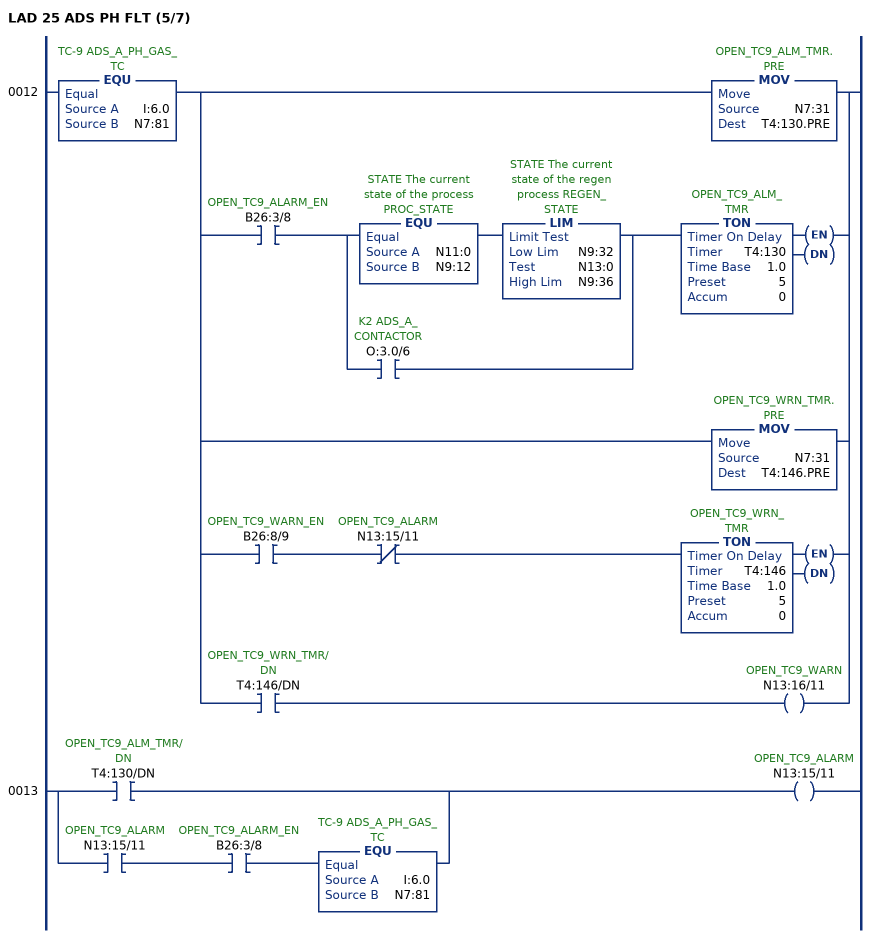
% Rung: 12 %
SOR EQU I:6.0 N7:81 BST MOV N7:31 T4:130.PRE NXB XIC B26:3/8 BST EQU N11:0 N9:12 LIM N9:32 N13:0 N9:36 NXB XIC O:3.0/6 BND TON T4:130 1.0 5 0 NXB MOV N7:31 T4:146.PRE NXB XIC B26:8/9 XIO N13:15/11 TON T4:146 1.0 5 0 NXB XIC T4:146/DN OTE N13:16/11 BND EOR
%   I:6.0  ADS_A_PH_GAS_TC  "TC-9" %
%   N7:81  TC_OPEN_SP  "CONFIG The value read by an open TC input" %
%   N7:31  OPEN_TC_DLY %
%   T4:130  OPEN_TC9_ALM_TMR %
%   B26:3/8  OPEN_TC9_ALARM_EN %
%   N11:0  PROC_STATE  "STATE The current state of the process" %
%   N9:12  PROC_PFY_B_REG_A  "STATE Process Purify B" %
%   N9:32  REGEN_VENT  "STATE Regen Vent" %
%   N13:0  REGEN_STATE  "STATE The current state of the regen process" %
%   N9:36  REGEN_COOL  "STATE Regen Cool" %
%   O:3.0/6  ADS_A_CONTACTOR  "K2" %
%   T4:146  OPEN_TC9_WRN_TMR %
%   B26:8/9  OPEN_TC9_WARN_EN %
%   N13:15/11  OPEN_TC9_ALARM %
%   N13:16/11  OPEN_TC9_WARN %
% Rung: 13 %
SOR BST XIC T4:130/DN NXB XIC N13:15/11 XIC B26:3/8 EQU I:6.0 N7:81 BND OTE N13:15/11 EOR
%   T4:130  OPEN_TC9_ALM_TMR %
%   N13:15/11  OPEN_TC9_ALARM %
%   B26:3/8  OPEN_TC9_ALARM_EN %
%   I:6.0  ADS_A_PH_GAS_TC  "TC-9" %
%   N7:81  TC_OPEN_SP  "CONFIG The value read by an open TC input" %

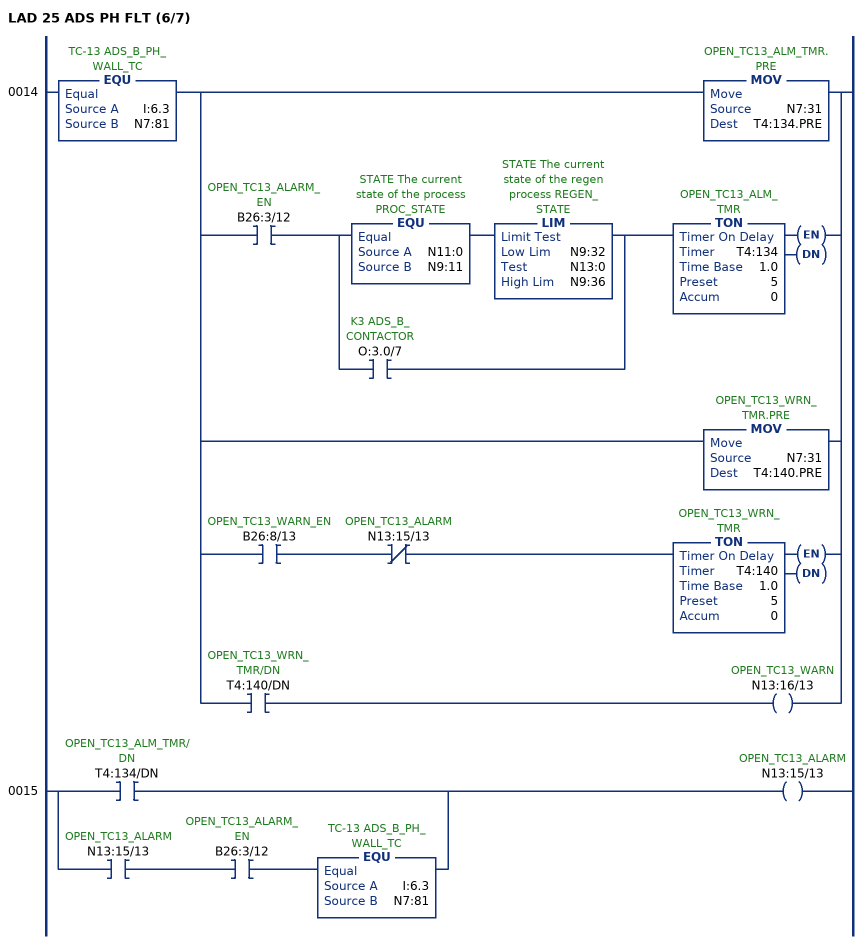
% Rung: 14 %
SOR EQU I:6.3 N7:81 BST MOV N7:31 T4:134.PRE NXB XIC B26:3/12 BST EQU N11:0 N9:11 LIM N9:32 N13:0 N9:36 NXB XIC O:3.0/7 BND TON T4:134 1.0 5 0 NXB MOV N7:31 T4:140.PRE NXB XIC B26:8/13 XIO N13:15/13 TON T4:140 1.0 5 0 NXB XIC T4:140/DN OTE N13:16/13 BND EOR
%   I:6.3  ADS_B_PH_WALL_TC  "TC-13" %
%   N7:81  TC_OPEN_SP  "CONFIG The value read by an open TC input" %
%   N7:31  OPEN_TC_DLY %
%   T4:134  OPEN_TC13_ALM_TMR %
%   B26:3/12  OPEN_TC13_ALARM_EN %
%   N11:0  PROC_STATE  "STATE The current state of the process" %
%   N9:11  PROC_PFY_A_REG_B  "STATE Process Purify A" %
%   N9:32  REGEN_VENT  "STATE Regen Vent" %
%   N13:0  REGEN_STATE  "STATE The current state of the regen process" %
%   N9:36  REGEN_COOL  "STATE Regen Cool" %
%   O:3.0/7  ADS_B_CONTACTOR  "K3" %
%   T4:140  OPEN_TC13_WRN_TMR %
%   B26:8/13  OPEN_TC13_WARN_EN %
%   N13:15/13  OPEN_TC13_ALARM %
%   N13:16/13  OPEN_TC13_WARN %
% Rung: 15 %
SOR BST XIC T4:134/DN NXB XIC N13:15/13 XIC B26:3/12 EQU I:6.3 N7:81 BND OTE N13:15/13 EOR
%   T4:134  OPEN_TC13_ALM_TMR %
%   N13:15/13  OPEN_TC13_ALARM %
%   B26:3/12  OPEN_TC13_ALARM_EN %
%   I:6.3  ADS_B_PH_WALL_TC  "TC-13" %
%   N7:81  TC_OPEN_SP  "CONFIG The value read by an open TC input" %

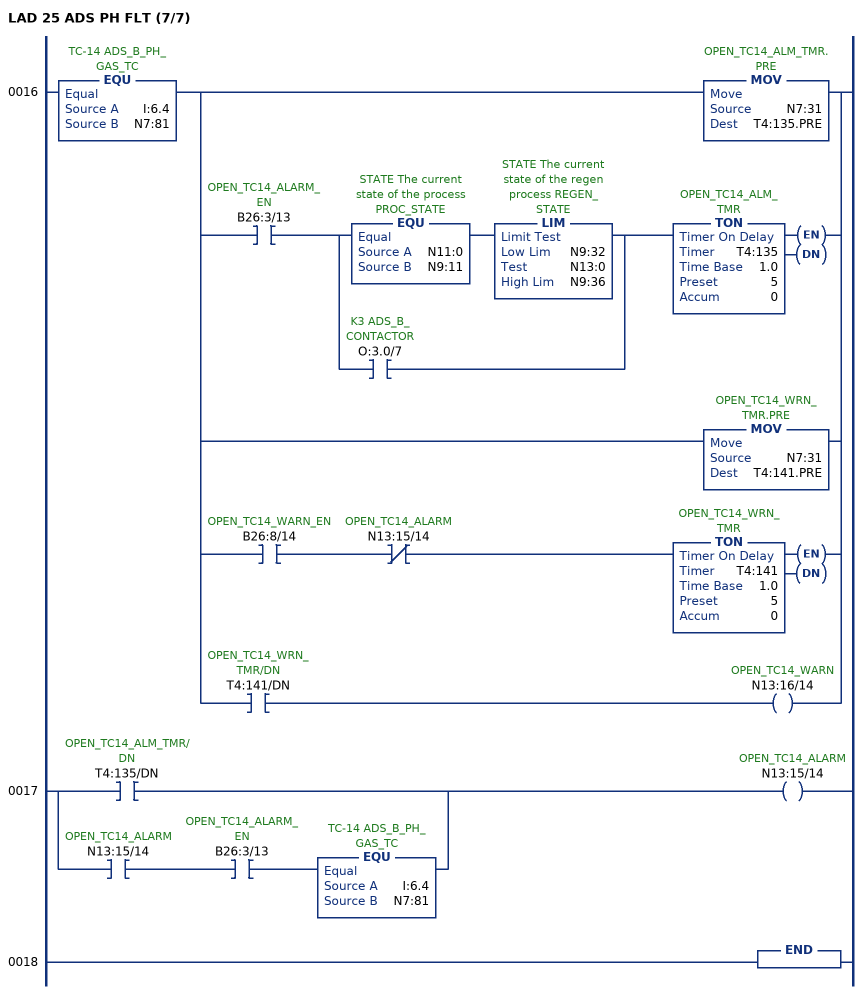
% Rung: 16 %
SOR EQU I:6.4 N7:81 BST MOV N7:31 T4:135.PRE NXB XIC B26:3/13 BST EQU N11:0 N9:11 LIM N9:32 N13:0 N9:36 NXB XIC O:3.0/7 BND TON T4:135 1.0 5 0 NXB MOV N7:31 T4:141.PRE NXB XIC B26:8/14 XIO N13:15/14 TON T4:141 1.0 5 0 NXB XIC T4:141/DN OTE N13:16/14 BND EOR
%   I:6.4  ADS_B_PH_GAS_TC  "TC-14" %
%   N7:81  TC_OPEN_SP  "CONFIG The value read by an open TC input" %
%   N7:31  OPEN_TC_DLY %
%   T4:135  OPEN_TC14_ALM_TMR %
%   B26:3/13  OPEN_TC14_ALARM_EN %
%   N11:0  PROC_STATE  "STATE The current state of the process" %
%   N9:11  PROC_PFY_A_REG_B  "STATE Process Purify A" %
%   N9:32  REGEN_VENT  "STATE Regen Vent" %
%   N13:0  REGEN_STATE  "STATE The current state of the regen process" %
%   N9:36  REGEN_COOL  "STATE Regen Cool" %
%   O:3.0/7  ADS_B_CONTACTOR  "K3" %
%   T4:141  OPEN_TC14_WRN_TMR %
%   B26:8/14  OPEN_TC14_WARN_EN %
%   N13:15/14  OPEN_TC14_ALARM %
%   N13:16/14  OPEN_TC14_WARN %
% Rung: 17 %
SOR BST XIC T4:135/DN NXB XIC N13:15/14 XIC B26:3/13 EQU I:6.4 N7:81 BND OTE N13:15/14 EOR
%   T4:135  OPEN_TC14_ALM_TMR %
%   N13:15/14  OPEN_TC14_ALARM %
%   B26:3/13  OPEN_TC14_ALARM_EN %
%   I:6.4  ADS_B_PH_GAS_TC  "TC-14" %
%   N7:81  TC_OPEN_SP  "CONFIG The value read by an open TC input" %
% Rung: 18 %
SOR END EOR

LADDER 26 "GETTER"
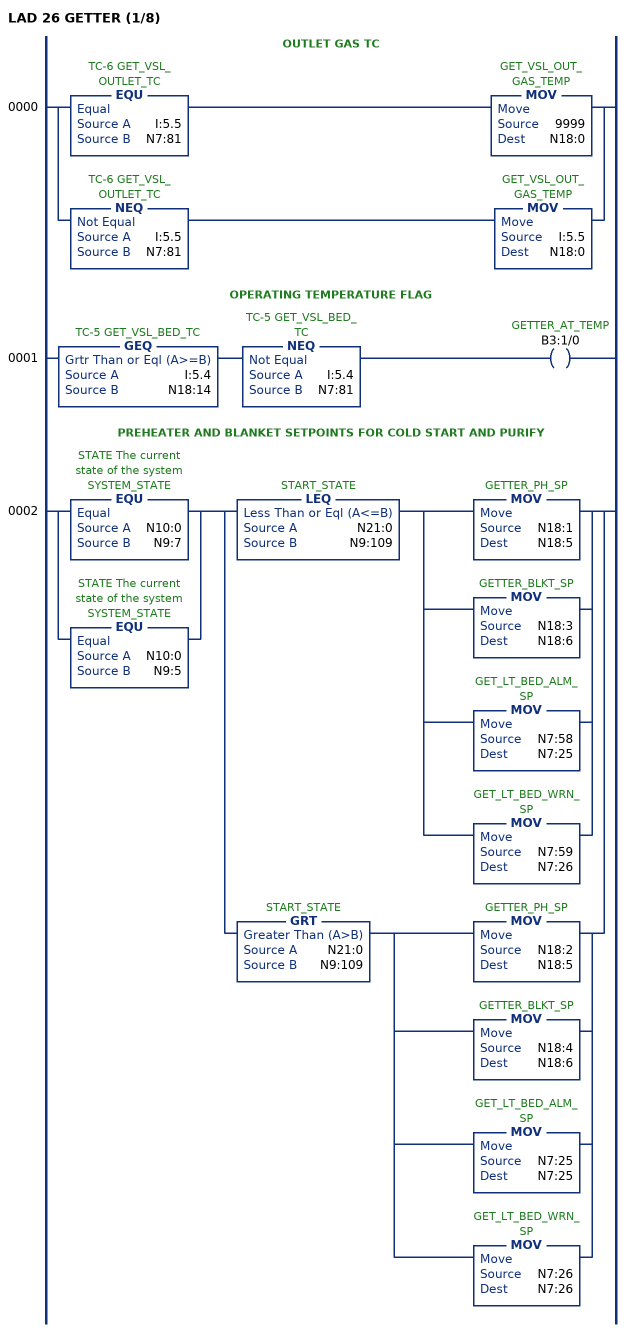
% Rung: 0 %
% TITLE: OUTLET GAS TC %
SOR BST EQU I:5.5 N7:81 MOV 9999 N18:0 NXB NEQ I:5.5 N7:81 MOV I:5.5 N18:0 BND EOR
%   I:5.5  GET_VSL_OUTLET_TC  "TC-6" %
%   N7:81  TC_OPEN_SP  "CONFIG The value read by an open TC input" %
%   N18:0  GET_VSL_OUT_GAS_TEMP %
% Rung: 1 %
% TITLE: OPERATING TEMPERATURE FLAG %
SOR GEQ I:5.4 N18:14 NEQ I:5.4 N7:81 OTE B3:1/0 EOR
%   I:5.4  GET_VSL_BED_TC  "TC-5" %
%   N18:14  GETTER_OPERATING_TMP %
%   N7:81  TC_OPEN_SP  "CONFIG The value read by an open TC input" %
%   B3:1/0  GETTER_AT_TEMP %
% Rung: 2 %
% TITLE: PREHEATER AND BLANKET SETPOINTS FOR COLD START AND PURIFY %
SOR BST EQU N10:0 N9:7 NXB EQU N10:0 N9:5 BND BST LEQ N21:0 N9:109 BST MOV N18:1 N18:5 NXB MOV N18:3 N18:6 NXB MOV N7:58 N7:25 NXB MOV N7:59 N7:26 BND NXB GRT N21:0 N9:109 BST MOV N18:2 N18:5 NXB MOV N18:4 N18:6 NXB MOV N7:25 N7:25 NXB MOV N7:26 N7:26 BND BND EOR
%   N10:0  SYSTEM_STATE  "STATE The current state of the system" %
%   N9:7  SYSTEM_COLD_START %
%   N9:5  SYSTEM_QUICK_START %
%   N21:0  START_STATE %
%   N9:109  START_BKFL_2 %
%   N18:1  GETTER_COLD_PH_SP %
%   N18:5  GETTER_PH_SP %
%   N18:3  GETTER_COLD_BLKT_SP %
%   N18:6  GETTER_BLKT_SP %
%   N7:58  GET_LT_BED_ST_ALM_SP %
%   N7:25  GET_LT_BED_ALM_SP %
%   N7:59  GET_LT_BED_ST_WRN_SP %
%   N7:26  GET_LT_BED_WRN_SP %
%   N18:2  GETTER_PFY_PH_SP %
%   N18:4  GETTER_PFY_BLKT_SP %

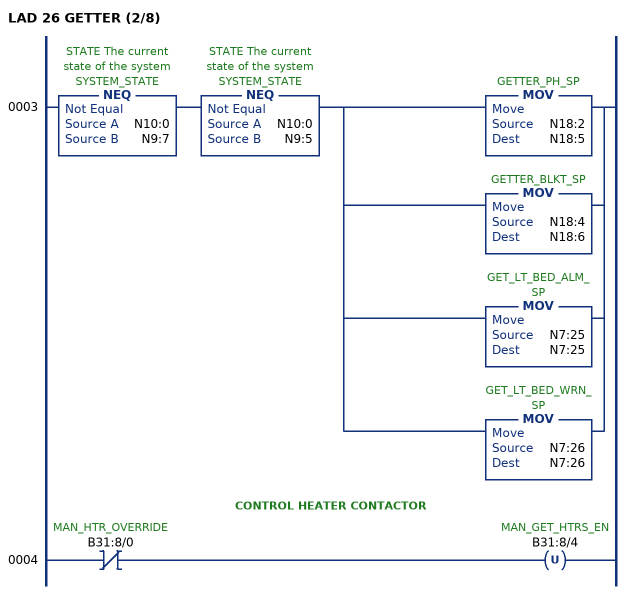
% Rung: 3 %
SOR NEQ N10:0 N9:7 NEQ N10:0 N9:5 BST MOV N18:2 N18:5 NXB MOV N18:4 N18:6 NXB MOV N7:25 N7:25 NXB MOV N7:26 N7:26 BND EOR
%   N10:0  SYSTEM_STATE  "STATE The current state of the system" %
%   N9:7  SYSTEM_COLD_START %
%   N9:5  SYSTEM_QUICK_START %
%   N18:2  GETTER_PFY_PH_SP %
%   N18:5  GETTER_PH_SP %
%   N18:4  GETTER_PFY_BLKT_SP %
%   N18:6  GETTER_BLKT_SP %
%   N7:25  GET_LT_BED_ALM_SP %
%   N7:26  GET_LT_BED_WRN_SP %
% Rung: 4 %
% TITLE: CONTROL HEATER CONTACTOR %
SOR XIO B31:8/0 OTU B31:8/4 EOR
%   B31:8/0  MAN_HTR_OVERRIDE %
%   B31:8/4  MAN_GET_HTRS_EN %

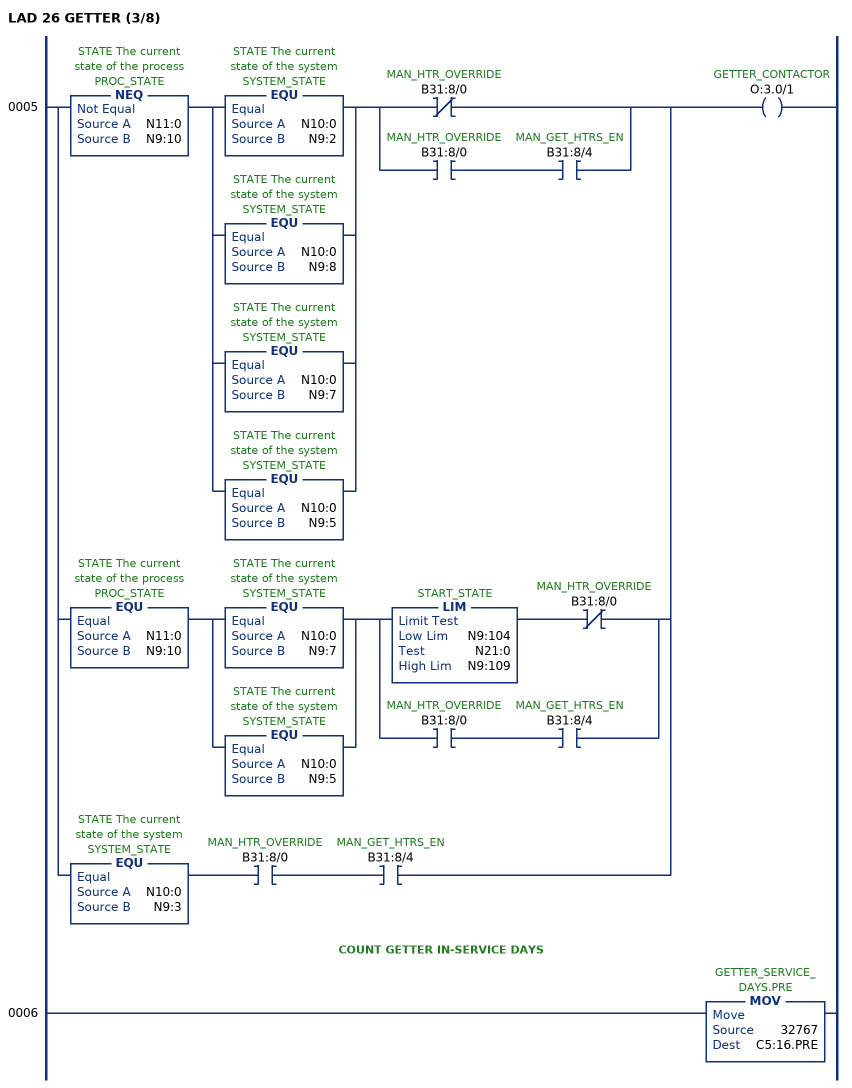
% Rung: 5 %
SOR BST NEQ N11:0 N9:10 BST EQU N10:0 N9:2 NXB EQU N10:0 N9:8 NXB EQU N10:0 N9:7 NXB EQU N10:0 N9:5 BND BST XIO B31:8/0 NXB XIC B31:8/0 XIC B31:8/4 BND NXB EQU N11:0 N9:10 BST EQU N10:0 N9:7 NXB EQU N10:0 N9:5 BND BST LIM N9:104 N21:0 N9:109 XIO B31:8/0 NXB XIC B31:8/0 XIC B31:8/4 BND NXB EQU N10:0 N9:3 XIC B31:8/0 XIC B31:8/4 BND OTE O:3.0/1 EOR
%   N11:0  PROC_STATE  "STATE The current state of the process" %
%   N9:10  PROC_STANDBY  "STATE Process Standby" %
%   N10:0  SYSTEM_STATE  "STATE The current state of the system" %
%   N9:2  SYSTEM_PROCESS  "STATE System Process" %
%   N9:8  SYSTEM_SUPPLEMENTAL %
%   N9:7  SYSTEM_COLD_START %
%   N9:5  SYSTEM_QUICK_START %
%   B31:8/0  MAN_HTR_OVERRIDE %
%   B31:8/4  MAN_GET_HTRS_EN %
%   N9:104  START_HEAT_GETTER %
%   N21:0  START_STATE %
%   N9:109  START_BKFL_2 %
%   N9:3  SYSTEM_MANUAL  "STATE System Manual" %
%   O:3.0/1  GETTER_CONTACTOR %
% Rung: 6 %
% TITLE: COUNT GETTER IN-SERVICE DAYS %
SOR MOV 32767 C5:16.PRE EOR
%   C5:16  GETTER_SERVICE_DAYS %

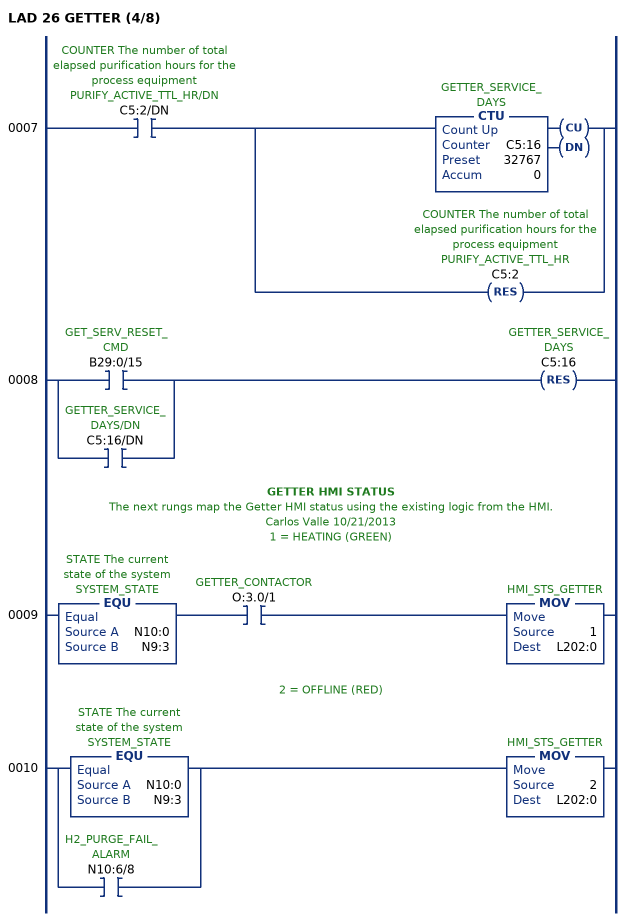
% Rung: 7 %
SOR XIC C5:2/DN BST CTU C5:16 32767 0 NXB RES C5:2 BND EOR
%   C5:2  PURIFY_ACTIVE_TTL_HR  "COUNTER The number of total elapsed purification hours for the process equipment" %
%   C5:16  GETTER_SERVICE_DAYS %
% Rung: 8 %
SOR BST XIC B29:0/15 NXB XIC C5:16/DN BND RES C5:16 EOR
%   B29:0/15  GET_SERV_RESET_CMD %
%   C5:16  GETTER_SERVICE_DAYS %
% Rung: 9 %
% TITLE: GETTER HMI STATUS %
% The next rungs map the Getter HMI status using the existing logic from the HMI.
% Carlos Valle 10/21/2013
% 1 = HEATING (GREEN) %
SOR EQU N10:0 N9:3 XIC O:3.0/1 MOV 1 L202:0 EOR
%   N10:0  SYSTEM_STATE  "STATE The current state of the system" %
%   N9:3  SYSTEM_MANUAL  "STATE System Manual" %
%   O:3.0/1  GETTER_CONTACTOR %
%   L202:0  HMI_STS_GETTER %
% Rung: 10 %
% 2 = OFFLINE (RED) %
SOR BST EQU N10:0 N9:3 NXB XIC N10:6/8 BND MOV 2 L202:0 EOR
%   N10:0  SYSTEM_STATE  "STATE The current state of the system" %
%   N9:3  SYSTEM_MANUAL  "STATE System Manual" %
%   N10:6/8  H2_PURGE_FAIL_ALARM %
%   L202:0  HMI_STS_GETTER %

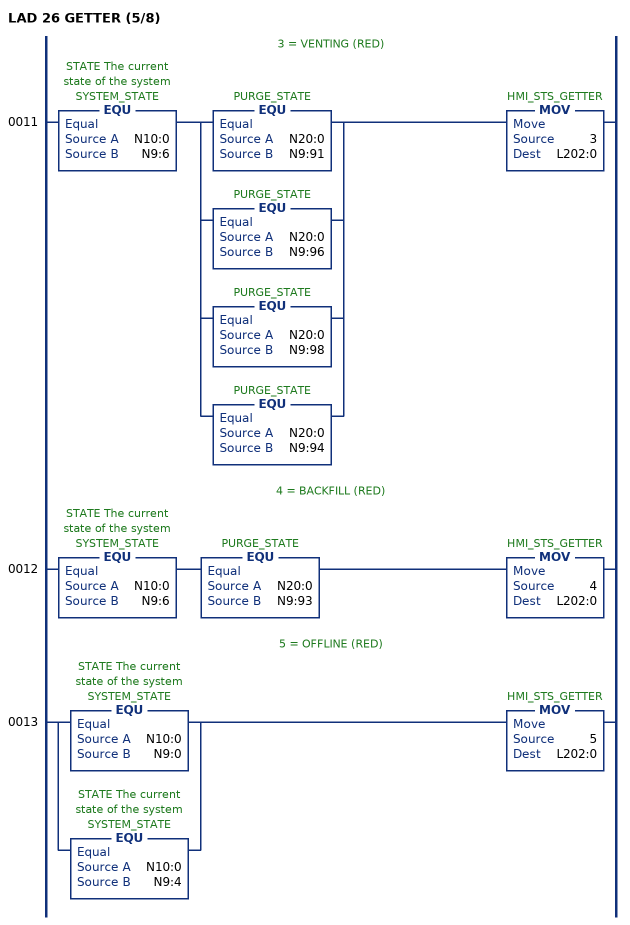
% Rung: 11 %
% 3 = VENTING (RED) %
SOR EQU N10:0 N9:6 BST EQU N20:0 N9:91 NXB EQU N20:0 N9:96 NXB EQU N20:0 N9:98 NXB EQU N20:0 N9:94 BND MOV 3 L202:0 EOR
%   N10:0  SYSTEM_STATE  "STATE The current state of the system" %
%   N9:6  SYSTEM_PURGE %
%   N20:0  PURGE_STATE %
%   N9:91  PURGE_INIT_VENT %
%   N9:96  PURGE_VENT_GETTER %
%   N9:98  PURGE_VENT_GET_2 %
%   N9:94  PURGE_FINAL_VENT %
%   L202:0  HMI_STS_GETTER %
% Rung: 12 %
% 4 = BACKFILL (RED) %
SOR EQU N10:0 N9:6 EQU N20:0 N9:93 MOV 4 L202:0 EOR
%   N10:0  SYSTEM_STATE  "STATE The current state of the system" %
%   N9:6  SYSTEM_PURGE %
%   N20:0  PURGE_STATE %
%   N9:93  PURGE_BACKFILL %
%   L202:0  HMI_STS_GETTER %
% Rung: 13 %
% 5 = OFFLINE (RED) %
SOR BST EQU N10:0 N9:0 NXB EQU N10:0 N9:4 BND MOV 5 L202:0 EOR
%   N10:0  SYSTEM_STATE  "STATE The current state of the system" %
%   N9:0  SYSTEM_OFFLINE %
%   N9:4  SYSTEM_ALARM  "STATE System Alarm" %
%   L202:0  HMI_STS_GETTER %

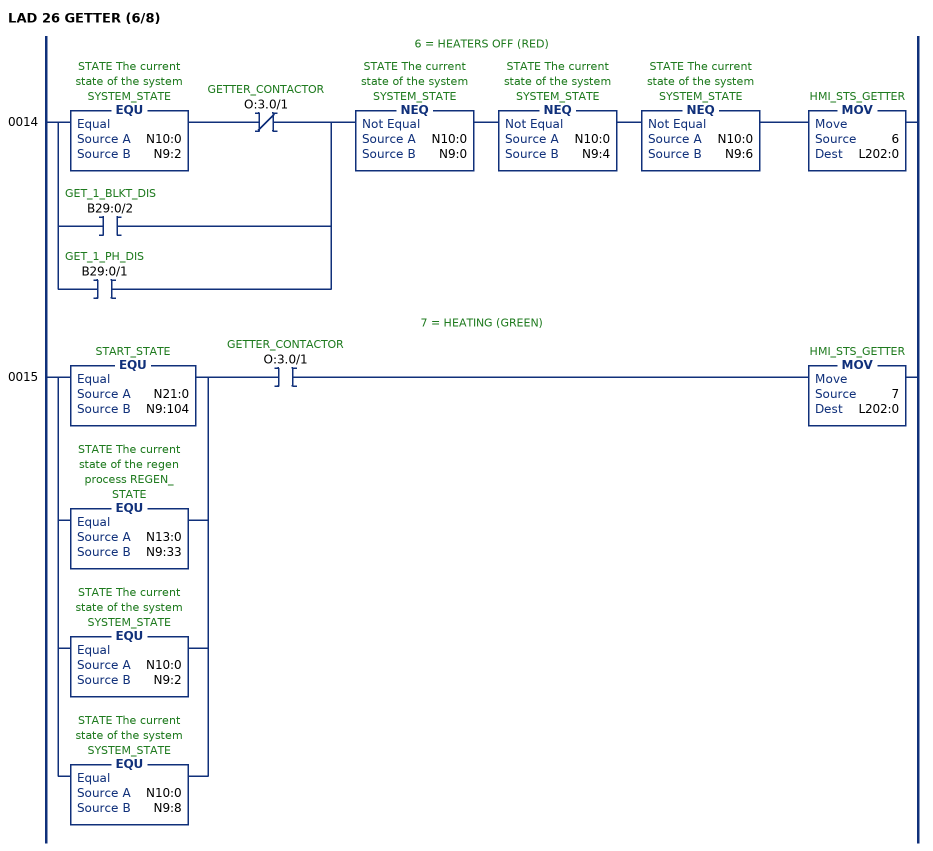
% Rung: 14 %
% 6 = HEATERS OFF (RED) %
SOR BST EQU N10:0 N9:2 XIO O:3.0/1 NXB XIC B29:0/2 NXB XIC B29:0/1 BND NEQ N10:0 N9:0 NEQ N10:0 N9:4 NEQ N10:0 N9:6 MOV 6 L202:0 EOR
%   N10:0  SYSTEM_STATE  "STATE The current state of the system" %
%   N9:2  SYSTEM_PROCESS  "STATE System Process" %
%   O:3.0/1  GETTER_CONTACTOR %
%   B29:0/2  GET_1_BLKT_DIS %
%   B29:0/1  GET_1_PH_DIS %
%   N9:0  SYSTEM_OFFLINE %
%   N9:4  SYSTEM_ALARM  "STATE System Alarm" %
%   N9:6  SYSTEM_PURGE %
%   L202:0  HMI_STS_GETTER %
% Rung: 15 %
% 7 = HEATING (GREEN) %
SOR BST EQU N21:0 N9:104 NXB EQU N13:0 N9:33 NXB EQU N10:0 N9:2 NXB EQU N10:0 N9:8 BND XIC O:3.0/1 MOV 7 L202:0 EOR
%   N21:0  START_STATE %
%   N9:104  START_HEAT_GETTER %
%   N13:0  REGEN_STATE  "STATE The current state of the regen process" %
%   N9:33  REGEN_HEAT_BED  "STATE Regen Heat wall" %
%   N10:0  SYSTEM_STATE  "STATE The current state of the system" %
%   N9:2  SYSTEM_PROCESS  "STATE System Process" %
%   N9:8  SYSTEM_SUPPLEMENTAL %
%   O:3.0/1  GETTER_CONTACTOR %
%   L202:0  HMI_STS_GETTER %

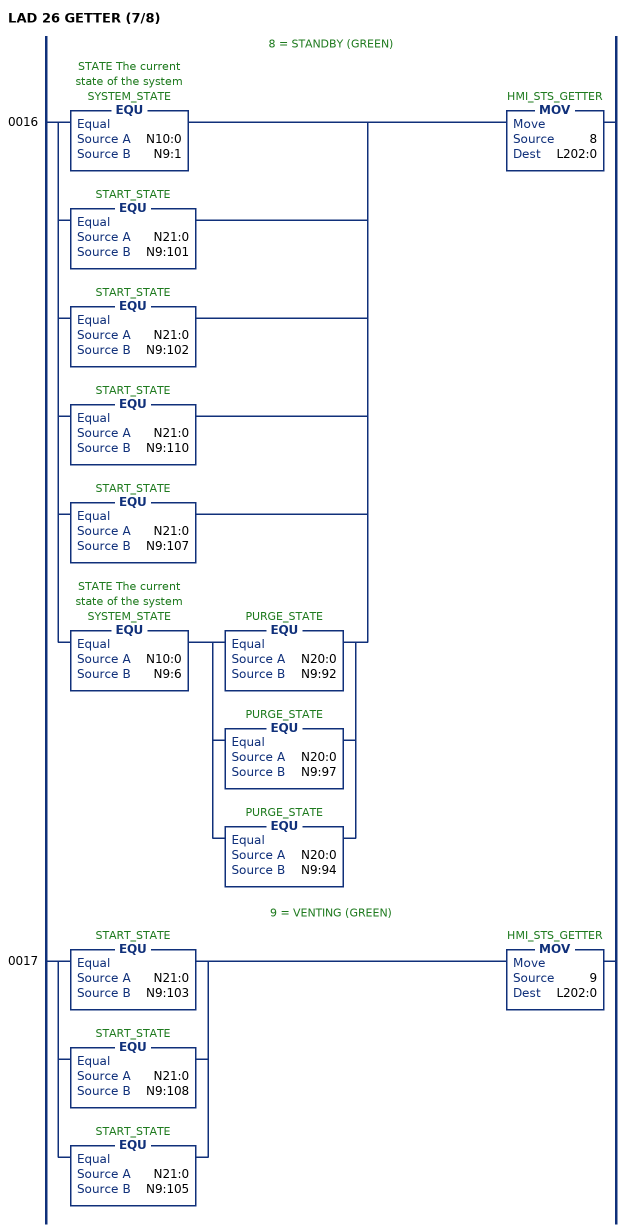
% Rung: 16 %
% 8 = STANDBY (GREEN) %
SOR BST EQU N10:0 N9:1 NXB EQU N21:0 N9:101 NXB EQU N21:0 N9:102 NXB EQU N21:0 N9:110 NXB EQU N21:0 N9:107 NXB EQU N10:0 N9:6 BST EQU N20:0 N9:92 NXB EQU N20:0 N9:97 NXB EQU N20:0 N9:94 BND BND MOV 8 L202:0 EOR
%   N10:0  SYSTEM_STATE  "STATE The current state of the system" %
%   N9:1  SYSTEM_STANDBY  "STATE System Process" %
%   N21:0  START_STATE %
%   N9:101  START_COOL %
%   N9:102  START_VENT_ADS_1 %
%   N9:110  START_REG_VENT %
%   N9:107  START_VENT_ADS_2 %
%   N9:6  SYSTEM_PURGE %
%   N20:0  PURGE_STATE %
%   N9:92  PURGE_VENT_ADSORBER %
%   N9:97  PURGE_VENT_ADS_2 %
%   N9:94  PURGE_FINAL_VENT %
%   L202:0  HMI_STS_GETTER %
% Rung: 17 %
% 9 = VENTING (GREEN) %
SOR BST EQU N21:0 N9:103 NXB EQU N21:0 N9:108 NXB EQU N21:0 N9:105 BND MOV 9 L202:0 EOR
%   N21:0  START_STATE %
%   N9:103  START_VENT_GET_1 %
%   N9:108  START_VENT_GET_2 %
%   N9:105  START_VENT_ALL %
%   L202:0  HMI_STS_GETTER %

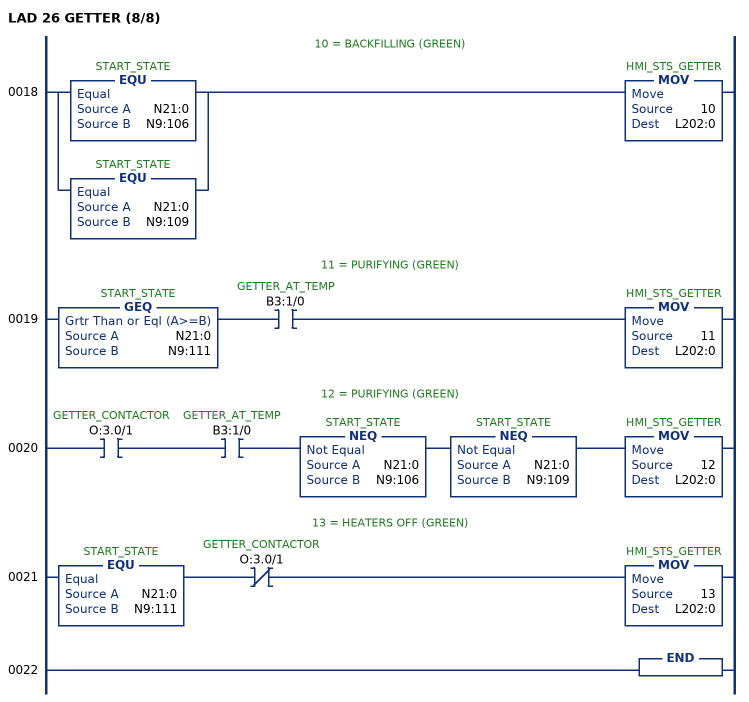
% Rung: 18 %
% 10 = BACKFILLING (GREEN) %
SOR BST EQU N21:0 N9:106 NXB EQU N21:0 N9:109 BND MOV 10 L202:0 EOR
%   N21:0  START_STATE %
%   N9:106  START_BACKFILL_1 %
%   N9:109  START_BKFL_2 %
%   L202:0  HMI_STS_GETTER %
% Rung: 19 %
% 11 = PURIFYING (GREEN) %
SOR GEQ N21:0 N9:111 XIC B3:1/0 MOV 11 L202:0 EOR
%   N21:0  START_STATE %
%   N9:111  START_REG_HEAT %
%   B3:1/0  GETTER_AT_TEMP %
%   L202:0  HMI_STS_GETTER %
% Rung: 20 %
% 12 = PURIFYING (GREEN) %
SOR XIC O:3.0/1 XIC B3:1/0 NEQ N21:0 N9:106 NEQ N21:0 N9:109 MOV 12 L202:0 EOR
%   O:3.0/1  GETTER_CONTACTOR %
%   B3:1/0  GETTER_AT_TEMP %
%   N21:0  START_STATE %
%   N9:106  START_BACKFILL_1 %
%   N9:109  START_BKFL_2 %
%   L202:0  HMI_STS_GETTER %
% Rung: 21 %
% 13 = HEATERS OFF (GREEN) %
SOR EQU N21:0 N9:111 XIO O:3.0/1 MOV 13 L202:0 EOR
%   N21:0  START_STATE %
%   N9:111  START_REG_HEAT %
%   O:3.0/1  GETTER_CONTACTOR %
%   L202:0  HMI_STS_GETTER %
% Rung: 22 %
SOR END EOR

LADDER 27 "GET 1 FLT"
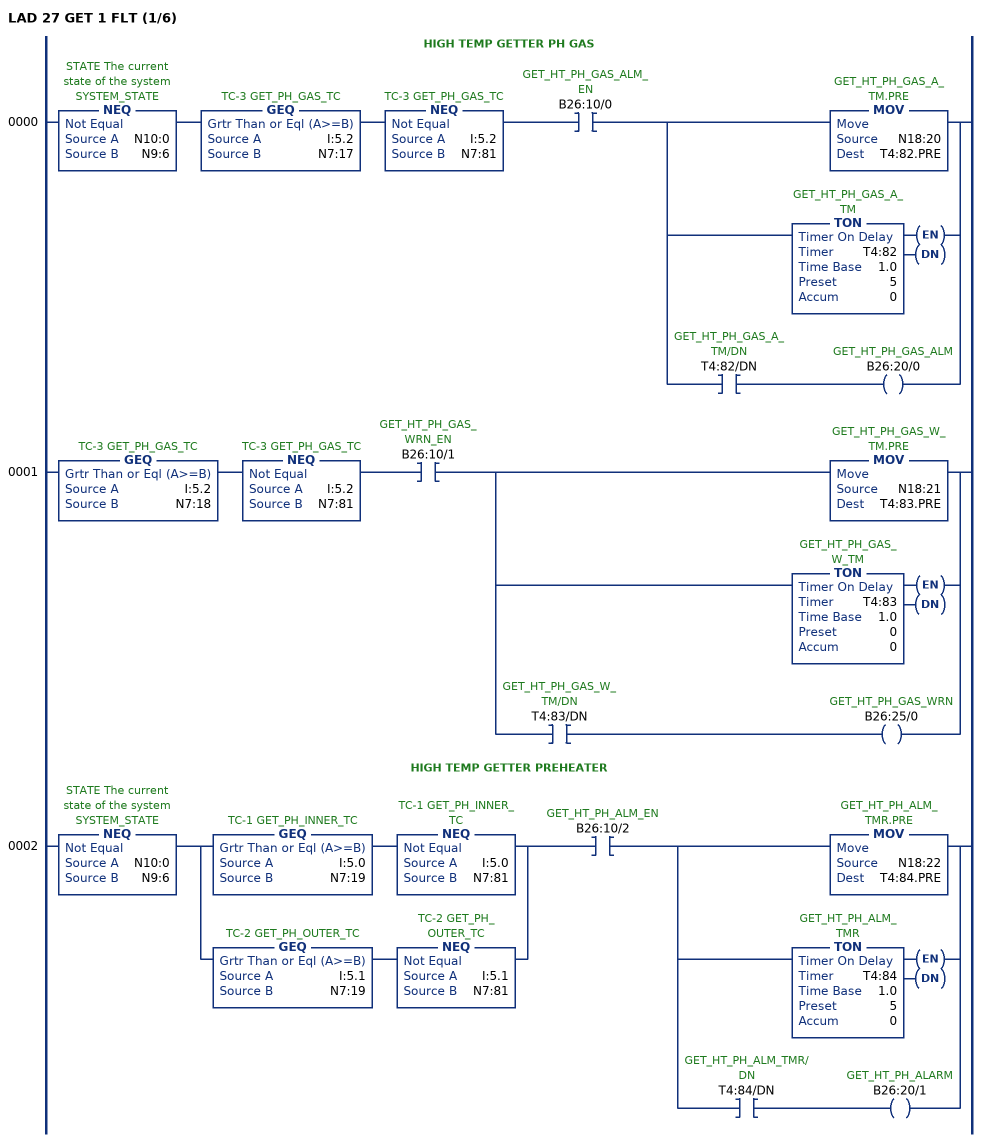
% Rung: 0 %
% TITLE: HIGH TEMP GETTER PH GAS %
SOR NEQ N10:0 N9:6 GEQ I:5.2 N7:17 NEQ I:5.2 N7:81 XIC B26:10/0 BST MOV N18:20 T4:82.PRE NXB TON T4:82 1.0 5 0 NXB XIC T4:82/DN OTE B26:20/0 BND EOR
%   N10:0  SYSTEM_STATE  "STATE The current state of the system" %
%   N9:6  SYSTEM_PURGE %
%   I:5.2  GET_PH_GAS_TC  "TC-3" %
%   N7:17  GET_HT_PH_GAS_ALM_SP %
%   N7:81  TC_OPEN_SP  "CONFIG The value read by an open TC input" %
%   B26:10/0  GET_HT_PH_GAS_ALM_EN %
%   N18:20  GET_HT_PH_GAS_ALM_DL %
%   T4:82  GET_HT_PH_GAS_A_TM %
%   B26:20/0  GET_HT_PH_GAS_ALM %
% Rung: 1 %
SOR GEQ I:5.2 N7:18 NEQ I:5.2 N7:81 XIC B26:10/1 BST MOV N18:21 T4:83.PRE NXB TON T4:83 1.0 0 0 NXB XIC T4:83/DN OTE B26:25/0 BND EOR
%   I:5.2  GET_PH_GAS_TC  "TC-3" %
%   N7:18  GET_HT_PH_GAS_WRN_SP %
%   N7:81  TC_OPEN_SP  "CONFIG The value read by an open TC input" %
%   B26:10/1  GET_HT_PH_GAS_WRN_EN %
%   N18:21  GET_HT_PH_GAS_WRN_DL %
%   T4:83  GET_HT_PH_GAS_W_TM %
%   B26:25/0  GET_HT_PH_GAS_WRN %
% Rung: 2 %
% TITLE: HIGH TEMP GETTER PREHEATER %
SOR NEQ N10:0 N9:6 BST GEQ I:5.0 N7:19 NEQ I:5.0 N7:81 NXB GEQ I:5.1 N7:19 NEQ I:5.1 N7:81 BND XIC B26:10/2 BST MOV N18:22 T4:84.PRE NXB TON T4:84 1.0 5 0 NXB XIC T4:84/DN OTE B26:20/1 BND EOR
%   N10:0  SYSTEM_STATE  "STATE The current state of the system" %
%   N9:6  SYSTEM_PURGE %
%   I:5.0  GET_PH_INNER_TC  "TC-1" %
%   N7:19  GET_HT_PH_ALM_SP %
%   N7:81  TC_OPEN_SP  "CONFIG The value read by an open TC input" %
%   I:5.1  GET_PH_OUTER_TC  "TC-2" %
%   B26:10/2  GET_HT_PH_ALM_EN %
%   N18:22  GET_HT_PH_ALM_DLY %
%   T4:84  GET_HT_PH_ALM_TMR %
%   B26:20/1  GET_HT_PH_ALARM %

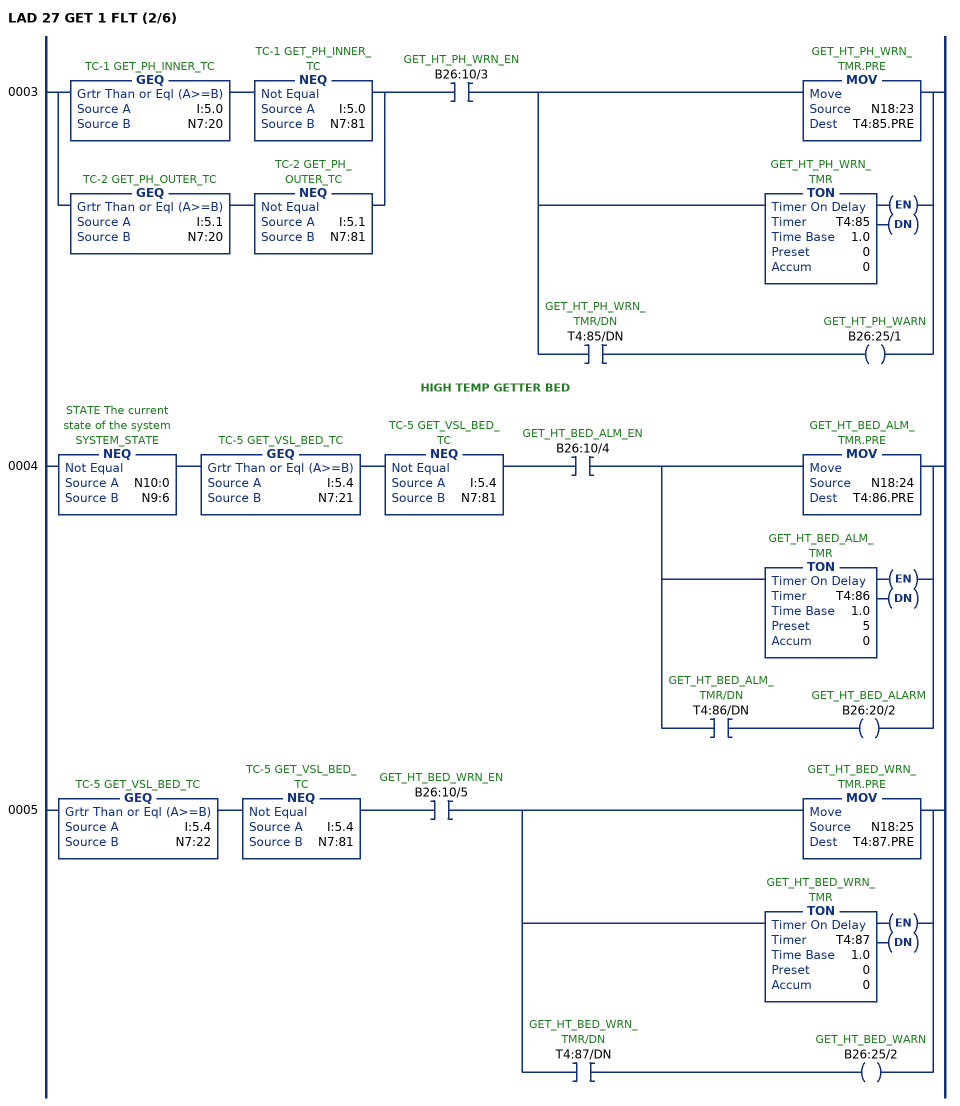
% Rung: 3 %
SOR BST GEQ I:5.0 N7:20 NEQ I:5.0 N7:81 NXB GEQ I:5.1 N7:20 NEQ I:5.1 N7:81 BND XIC B26:10/3 BST MOV N18:23 T4:85.PRE NXB TON T4:85 1.0 0 0 NXB XIC T4:85/DN OTE B26:25/1 BND EOR
%   I:5.0  GET_PH_INNER_TC  "TC-1" %
%   N7:20  GET_HT_PH_WRN_SP %
%   N7:81  TC_OPEN_SP  "CONFIG The value read by an open TC input" %
%   I:5.1  GET_PH_OUTER_TC  "TC-2" %
%   B26:10/3  GET_HT_PH_WRN_EN %
%   N18:23  GET_HT_PH_WRN_DLY %
%   T4:85  GET_HT_PH_WRN_TMR %
%   B26:25/1  GET_HT_PH_WARN %
% Rung: 4 %
% TITLE: HIGH TEMP GETTER BED %
SOR NEQ N10:0 N9:6 GEQ I:5.4 N7:21 NEQ I:5.4 N7:81 XIC B26:10/4 BST MOV N18:24 T4:86.PRE NXB TON T4:86 1.0 5 0 NXB XIC T4:86/DN OTE B26:20/2 BND EOR
%   N10:0  SYSTEM_STATE  "STATE The current state of the system" %
%   N9:6  SYSTEM_PURGE %
%   I:5.4  GET_VSL_BED_TC  "TC-5" %
%   N7:21  GET_HT_BED_ALM_SP %
%   N7:81  TC_OPEN_SP  "CONFIG The value read by an open TC input" %
%   B26:10/4  GET_HT_BED_ALM_EN %
%   N18:24  GET_HT_BED_ALM_DLY %
%   T4:86  GET_HT_BED_ALM_TMR %
%   B26:20/2  GET_HT_BED_ALARM %
% Rung: 5 %
SOR GEQ I:5.4 N7:22 NEQ I:5.4 N7:81 XIC B26:10/5 BST MOV N18:25 T4:87.PRE NXB TON T4:87 1.0 0 0 NXB XIC T4:87/DN OTE B26:25/2 BND EOR
%   I:5.4  GET_VSL_BED_TC  "TC-5" %
%   N7:22  GET_HT_BED_WRN_SP %
%   N7:81  TC_OPEN_SP  "CONFIG The value read by an open TC input" %
%   B26:10/5  GET_HT_BED_WRN_EN %
%   N18:25  GET_HT_BED_WRN_DLY %
%   T4:87  GET_HT_BED_WRN_TMR %
%   B26:25/2  GET_HT_BED_WARN %

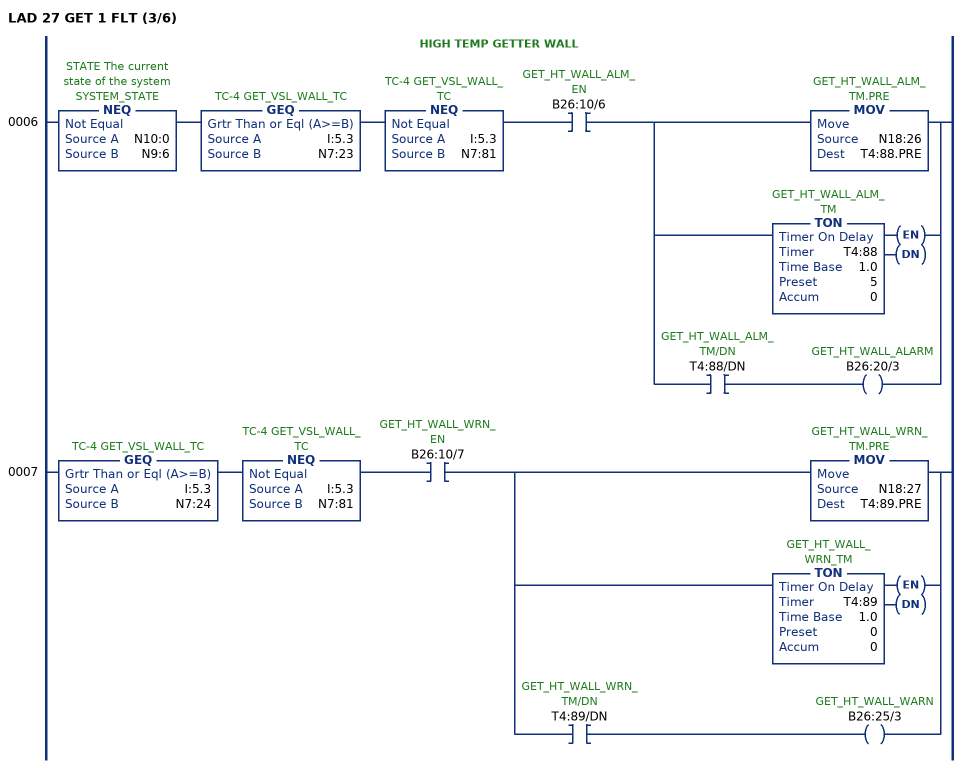
% Rung: 6 %
% TITLE: HIGH TEMP GETTER WALL %
SOR NEQ N10:0 N9:6 GEQ I:5.3 N7:23 NEQ I:5.3 N7:81 XIC B26:10/6 BST MOV N18:26 T4:88.PRE NXB TON T4:88 1.0 5 0 NXB XIC T4:88/DN OTE B26:20/3 BND EOR
%   N10:0  SYSTEM_STATE  "STATE The current state of the system" %
%   N9:6  SYSTEM_PURGE %
%   I:5.3  GET_VSL_WALL_TC  "TC-4" %
%   N7:23  GET_HT_WALL_ALM_SP %
%   N7:81  TC_OPEN_SP  "CONFIG The value read by an open TC input" %
%   B26:10/6  GET_HT_WALL_ALM_EN %
%   N18:26  GET_HT_WALL_ALM_DLY %
%   T4:88  GET_HT_WALL_ALM_TM %
%   B26:20/3  GET_HT_WALL_ALARM %
% Rung: 7 %
SOR GEQ I:5.3 N7:24 NEQ I:5.3 N7:81 XIC B26:10/7 BST MOV N18:27 T4:89.PRE NXB TON T4:89 1.0 0 0 NXB XIC T4:89/DN OTE B26:25/3 BND EOR
%   I:5.3  GET_VSL_WALL_TC  "TC-4" %
%   N7:24  GET_HT_WALL_WRN_SP %
%   N7:81  TC_OPEN_SP  "CONFIG The value read by an open TC input" %
%   B26:10/7  GET_HT_WALL_WRN_EN %
%   N18:27  GET_HT_WALL_WRN_DLY %
%   T4:89  GET_HT_WALL_WRN_TM %
%   B26:25/3  GET_HT_WALL_WARN %

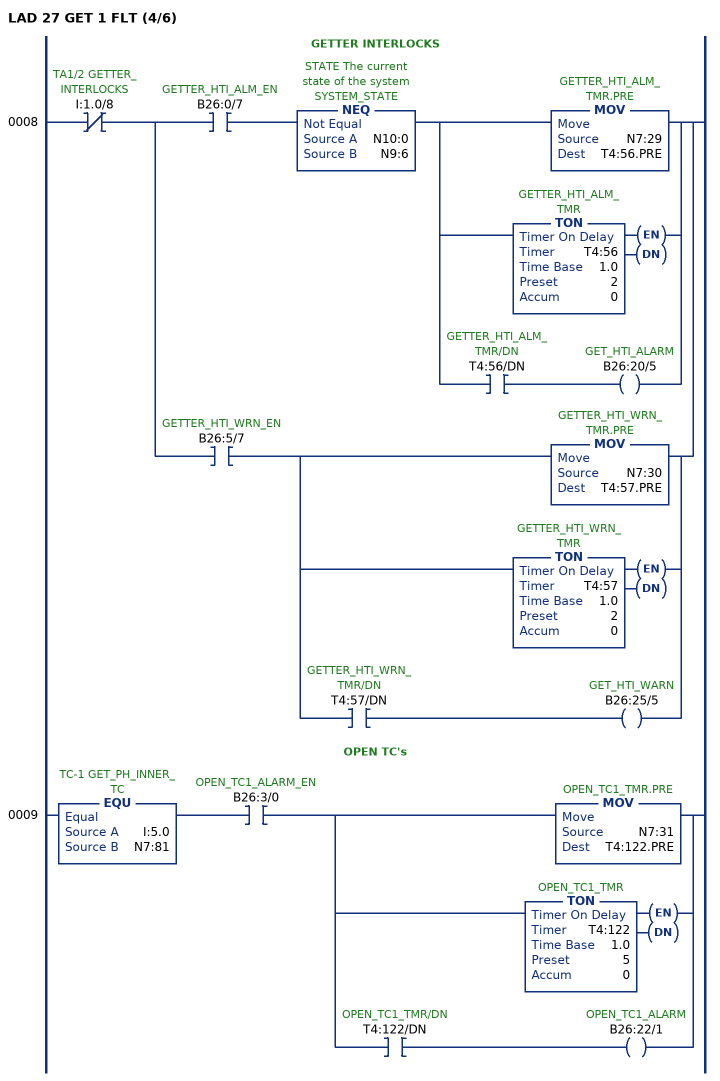
% Rung: 8 %
% TITLE: GETTER INTERLOCKS %
SOR XIO I:1.0/8 BST XIC B26:0/7 NEQ N10:0 N9:6 BST MOV N7:29 T4:56.PRE NXB TON T4:56 1.0 2 0 NXB XIC T4:56/DN OTE B26:20/5 BND NXB XIC B26:5/7 BST MOV N7:30 T4:57.PRE NXB TON T4:57 1.0 2 0 NXB XIC T4:57/DN OTE B26:25/5 BND BND EOR
%   I:1.0/8  GETTER_INTERLOCKS  "TA1/2" %
%   B26:0/7  GETTER_HTI_ALM_EN %
%   N10:0  SYSTEM_STATE  "STATE The current state of the system" %
%   N9:6  SYSTEM_PURGE %
%   N7:29  GETTER_HTI_ALM_DLY %
%   T4:56  GETTER_HTI_ALM_TMR %
%   B26:20/5  GET_HTI_ALARM %
%   B26:5/7  GETTER_HTI_WRN_EN %
%   N7:30  GETTER_HTI_WRN_DLY %
%   T4:57  GETTER_HTI_WRN_TMR %
%   B26:25/5  GET_HTI_WARN %
% Rung: 9 %
% TITLE: OPEN TC's %
SOR EQU I:5.0 N7:81 XIC B26:3/0 BST MOV N7:31 T4:122.PRE NXB TON T4:122 1.0 5 0 NXB XIC T4:122/DN OTE B26:22/1 BND EOR
%   I:5.0  GET_PH_INNER_TC  "TC-1" %
%   N7:81  TC_OPEN_SP  "CONFIG The value read by an open TC input" %
%   B26:3/0  OPEN_TC1_ALARM_EN %
%   N7:31  OPEN_TC_DLY %
%   T4:122  OPEN_TC1_TMR %
%   B26:22/1  OPEN_TC1_ALARM %

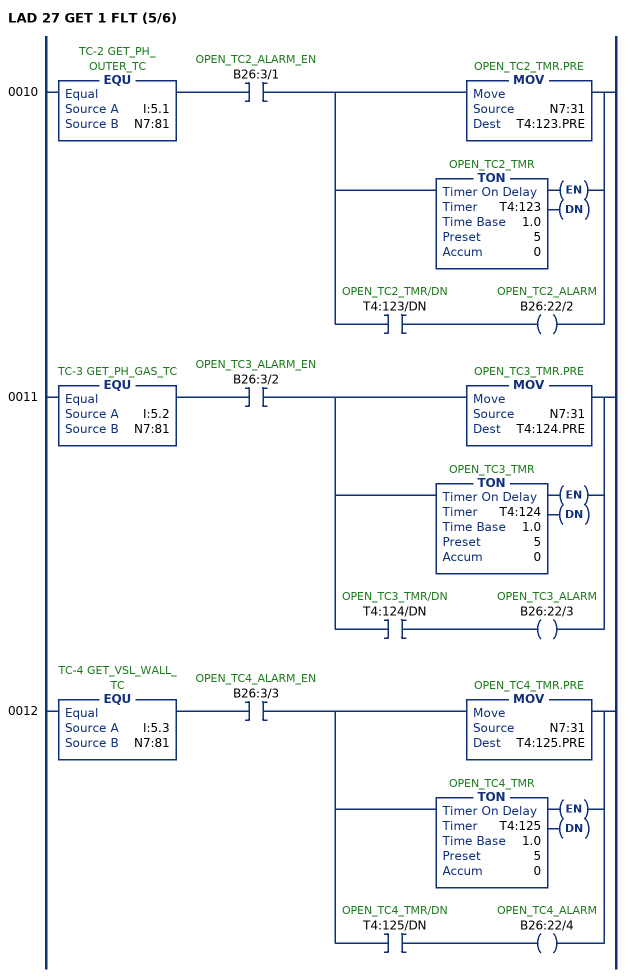
% Rung: 10 %
SOR EQU I:5.1 N7:81 XIC B26:3/1 BST MOV N7:31 T4:123.PRE NXB TON T4:123 1.0 5 0 NXB XIC T4:123/DN OTE B26:22/2 BND EOR
%   I:5.1  GET_PH_OUTER_TC  "TC-2" %
%   N7:81  TC_OPEN_SP  "CONFIG The value read by an open TC input" %
%   B26:3/1  OPEN_TC2_ALARM_EN %
%   N7:31  OPEN_TC_DLY %
%   T4:123  OPEN_TC2_TMR %
%   B26:22/2  OPEN_TC2_ALARM %
% Rung: 11 %
SOR EQU I:5.2 N7:81 XIC B26:3/2 BST MOV N7:31 T4:124.PRE NXB TON T4:124 1.0 5 0 NXB XIC T4:124/DN OTE B26:22/3 BND EOR
%   I:5.2  GET_PH_GAS_TC  "TC-3" %
%   N7:81  TC_OPEN_SP  "CONFIG The value read by an open TC input" %
%   B26:3/2  OPEN_TC3_ALARM_EN %
%   N7:31  OPEN_TC_DLY %
%   T4:124  OPEN_TC3_TMR %
%   B26:22/3  OPEN_TC3_ALARM %
% Rung: 12 %
SOR EQU I:5.3 N7:81 XIC B26:3/3 BST MOV N7:31 T4:125.PRE NXB TON T4:125 1.0 5 0 NXB XIC T4:125/DN OTE B26:22/4 BND EOR
%   I:5.3  GET_VSL_WALL_TC  "TC-4" %
%   N7:81  TC_OPEN_SP  "CONFIG The value read by an open TC input" %
%   B26:3/3  OPEN_TC4_ALARM_EN %
%   N7:31  OPEN_TC_DLY %
%   T4:125  OPEN_TC4_TMR %
%   B26:22/4  OPEN_TC4_ALARM %

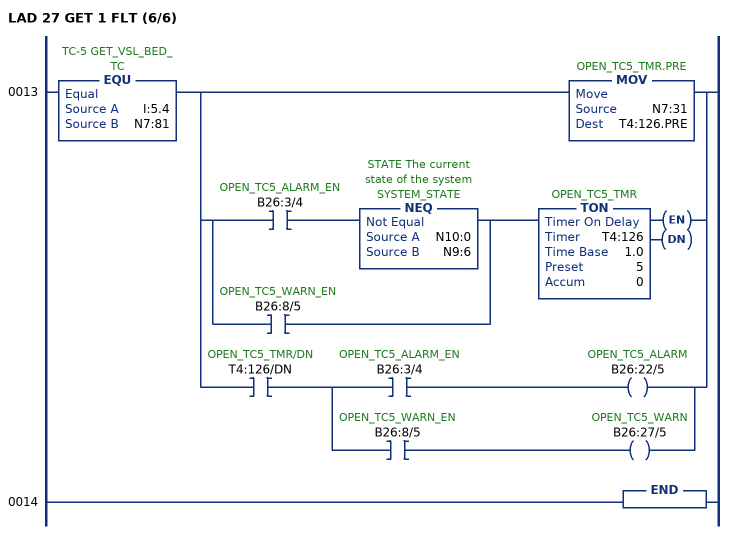
% Rung: 13 %
SOR EQU I:5.4 N7:81 BST MOV N7:31 T4:126.PRE NXB BST XIC B26:3/4 NEQ N10:0 N9:6 NXB XIC B26:8/5 BND TON T4:126 1.0 5 0 NXB XIC T4:126/DN BST XIC B26:3/4 OTE B26:22/5 NXB XIC B26:8/5 OTE B26:27/5 BND BND EOR
%   I:5.4  GET_VSL_BED_TC  "TC-5" %
%   N7:81  TC_OPEN_SP  "CONFIG The value read by an open TC input" %
%   N7:31  OPEN_TC_DLY %
%   T4:126  OPEN_TC5_TMR %
%   B26:3/4  OPEN_TC5_ALARM_EN %
%   N10:0  SYSTEM_STATE  "STATE The current state of the system" %
%   N9:6  SYSTEM_PURGE %
%   B26:8/5  OPEN_TC5_WARN_EN %
%   B26:22/5  OPEN_TC5_ALARM %
%   B26:27/5  OPEN_TC5_WARN %
% Rung: 14 %
SOR END EOR

LADDER 28 "GET 1"
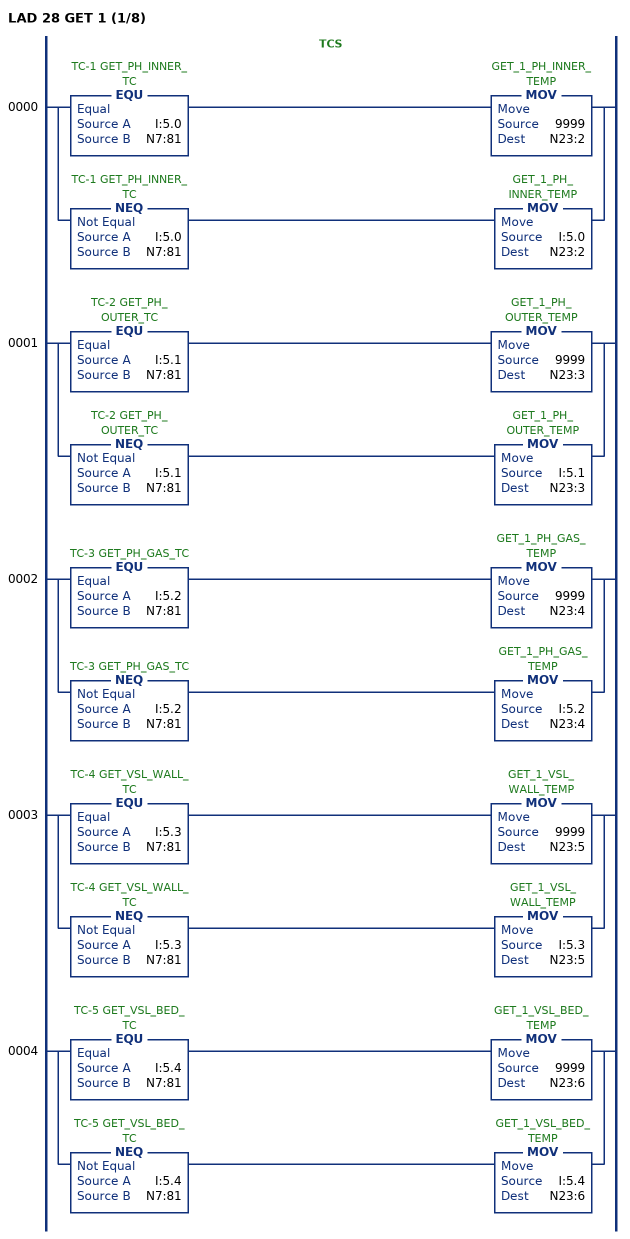
% Rung: 0 %
% TITLE: TCS %
SOR BST EQU I:5.0 N7:81 MOV 9999 N23:2 NXB NEQ I:5.0 N7:81 MOV I:5.0 N23:2 BND EOR
%   I:5.0  GET_PH_INNER_TC  "TC-1" %
%   N7:81  TC_OPEN_SP  "CONFIG The value read by an open TC input" %
%   N23:2  GET_1_PH_INNER_TEMP %
% Rung: 1 %
SOR BST EQU I:5.1 N7:81 MOV 9999 N23:3 NXB NEQ I:5.1 N7:81 MOV I:5.1 N23:3 BND EOR
%   I:5.1  GET_PH_OUTER_TC  "TC-2" %
%   N7:81  TC_OPEN_SP  "CONFIG The value read by an open TC input" %
%   N23:3  GET_1_PH_OUTER_TEMP %
% Rung: 2 %
SOR BST EQU I:5.2 N7:81 MOV 9999 N23:4 NXB NEQ I:5.2 N7:81 MOV I:5.2 N23:4 BND EOR
%   I:5.2  GET_PH_GAS_TC  "TC-3" %
%   N7:81  TC_OPEN_SP  "CONFIG The value read by an open TC input" %
%   N23:4  GET_1_PH_GAS_TEMP %
% Rung: 3 %
SOR BST EQU I:5.3 N7:81 MOV 9999 N23:5 NXB NEQ I:5.3 N7:81 MOV I:5.3 N23:5 BND EOR
%   I:5.3  GET_VSL_WALL_TC  "TC-4" %
%   N7:81  TC_OPEN_SP  "CONFIG The value read by an open TC input" %
%   N23:5  GET_1_VSL_WALL_TEMP %
% Rung: 4 %
SOR BST EQU I:5.4 N7:81 MOV 9999 N23:6 NXB NEQ I:5.4 N7:81 MOV I:5.4 N23:6 BND EOR
%   I:5.4  GET_VSL_BED_TC  "TC-5" %
%   N7:81  TC_OPEN_SP  "CONFIG The value read by an open TC input" %
%   N23:6  GET_1_VSL_BED_TEMP %

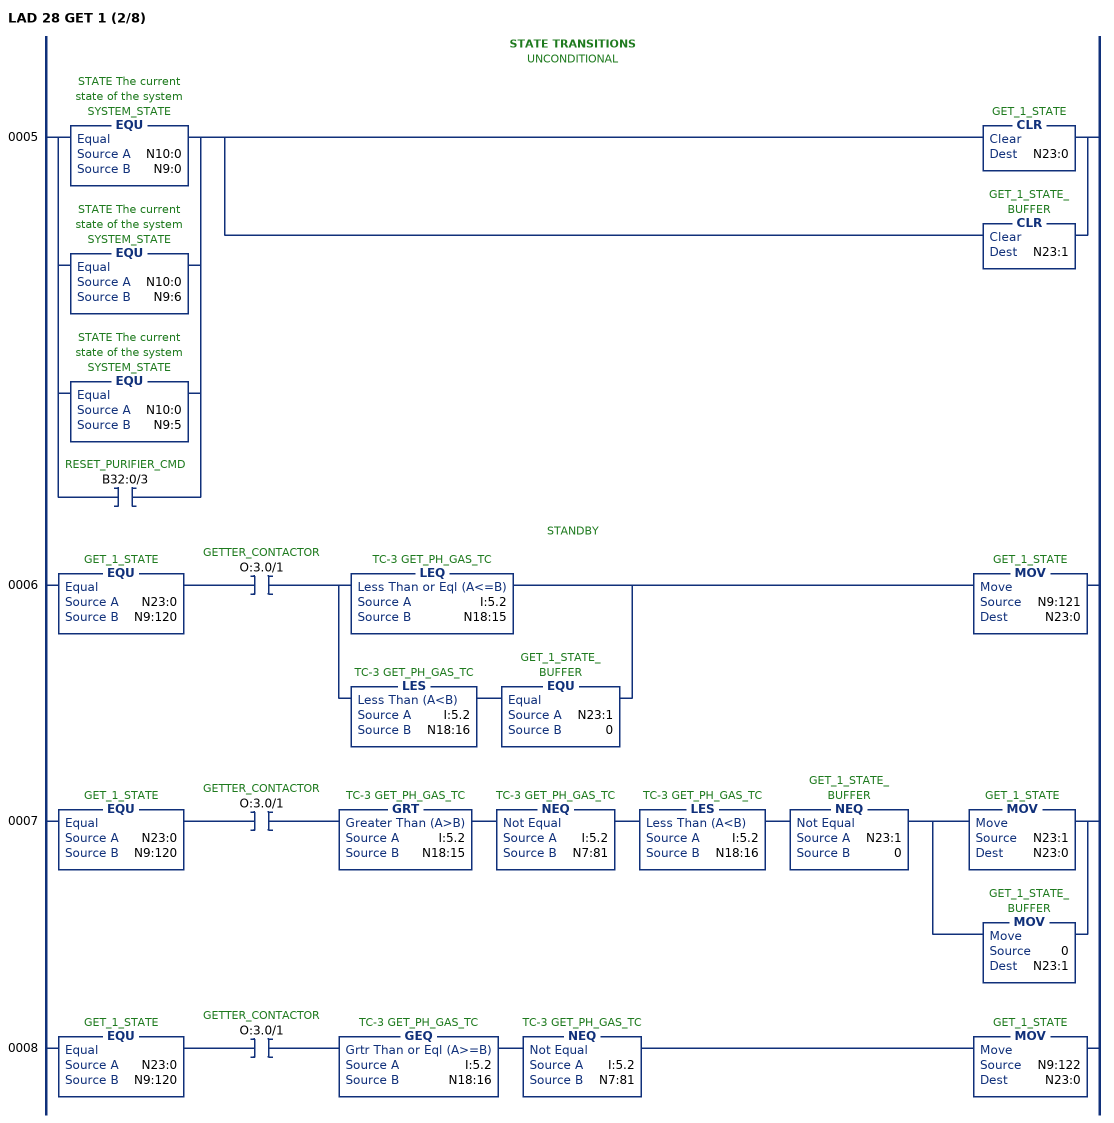
% Rung: 5 %
% TITLE: STATE TRANSITIONS %
% UNCONDITIONAL %
SOR BST EQU N10:0 N9:0 NXB EQU N10:0 N9:6 NXB EQU N10:0 N9:5 NXB XIC B32:0/3 BND BST CLR N23:0 NXB CLR N23:1 BND EOR
%   N10:0  SYSTEM_STATE  "STATE The current state of the system" %
%   N9:0  SYSTEM_OFFLINE %
%   N9:6  SYSTEM_PURGE %
%   N9:5  SYSTEM_QUICK_START %
%   B32:0/3  RESET_PURIFIER_CMD %
%   N23:0  GET_1_STATE %
%   N23:1  GET_1_STATE_BUFFER %
% Rung: 6 %
% STANDBY %
SOR EQU N23:0 N9:120 XIC O:3.0/1 BST LEQ I:5.2 N18:15 NXB LES I:5.2 N18:16 EQU N23:1 0 BND MOV N9:121 N23:0 EOR
%   N23:0  GET_1_STATE %
%   N9:120  GETTER_STANDBY %
%   O:3.0/1  GETTER_CONTACTOR %
%   I:5.2  GET_PH_GAS_TC  "TC-3" %
%   N18:15  GETTER_SS_BEGIN_TEMP %
%   N18:16  GETTER_SS_END_TEMP %
%   N23:1  GET_1_STATE_BUFFER %
%   N9:121  GETTER_SOFTSTART %
% Rung: 7 %
SOR EQU N23:0 N9:120 XIC O:3.0/1 GRT I:5.2 N18:15 NEQ I:5.2 N7:81 LES I:5.2 N18:16 NEQ N23:1 0 BST MOV N23:1 N23:0 NXB MOV 0 N23:1 BND EOR
%   N23:0  GET_1_STATE %
%   N9:120  GETTER_STANDBY %
%   O:3.0/1  GETTER_CONTACTOR %
%   I:5.2  GET_PH_GAS_TC  "TC-3" %
%   N18:15  GETTER_SS_BEGIN_TEMP %
%   N7:81  TC_OPEN_SP  "CONFIG The value read by an open TC input" %
%   N18:16  GETTER_SS_END_TEMP %
%   N23:1  GET_1_STATE_BUFFER %
% Rung: 8 %
SOR EQU N23:0 N9:120 XIC O:3.0/1 GEQ I:5.2 N18:16 NEQ I:5.2 N7:81 MOV N9:122 N23:0 EOR
%   N23:0  GET_1_STATE %
%   N9:120  GETTER_STANDBY %
%   O:3.0/1  GETTER_CONTACTOR %
%   I:5.2  GET_PH_GAS_TC  "TC-3" %
%   N18:16  GETTER_SS_END_TEMP %
%   N7:81  TC_OPEN_SP  "CONFIG The value read by an open TC input" %
%   N9:122  GETTER_PURIFYING %

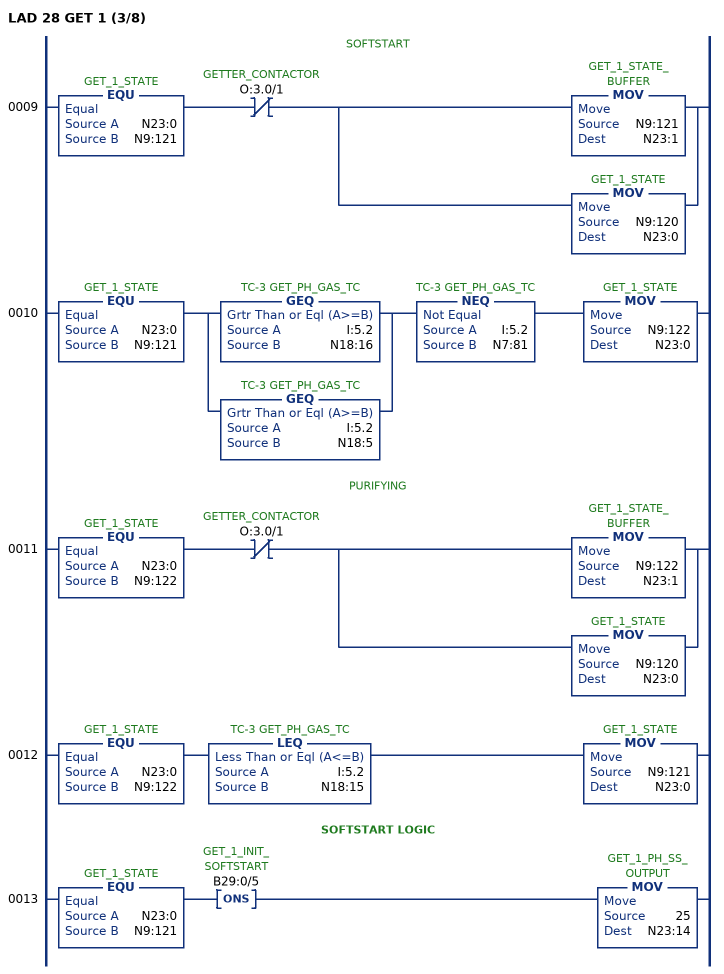
% Rung: 9 %
% SOFTSTART %
SOR EQU N23:0 N9:121 XIO O:3.0/1 BST MOV N9:121 N23:1 NXB MOV N9:120 N23:0 BND EOR
%   N23:0  GET_1_STATE %
%   N9:121  GETTER_SOFTSTART %
%   O:3.0/1  GETTER_CONTACTOR %
%   N23:1  GET_1_STATE_BUFFER %
%   N9:120  GETTER_STANDBY %
% Rung: 10 %
SOR EQU N23:0 N9:121 BST GEQ I:5.2 N18:16 NXB GEQ I:5.2 N18:5 BND NEQ I:5.2 N7:81 MOV N9:122 N23:0 EOR
%   N23:0  GET_1_STATE %
%   N9:121  GETTER_SOFTSTART %
%   I:5.2  GET_PH_GAS_TC  "TC-3" %
%   N18:16  GETTER_SS_END_TEMP %
%   N18:5  GETTER_PH_SP %
%   N7:81  TC_OPEN_SP  "CONFIG The value read by an open TC input" %
%   N9:122  GETTER_PURIFYING %
% Rung: 11 %
% PURIFYING %
SOR EQU N23:0 N9:122 XIO O:3.0/1 BST MOV N9:122 N23:1 NXB MOV N9:120 N23:0 BND EOR
%   N23:0  GET_1_STATE %
%   N9:122  GETTER_PURIFYING %
%   O:3.0/1  GETTER_CONTACTOR %
%   N23:1  GET_1_STATE_BUFFER %
%   N9:120  GETTER_STANDBY %
% Rung: 12 %
SOR EQU N23:0 N9:122 LEQ I:5.2 N18:15 MOV N9:121 N23:0 EOR
%   N23:0  GET_1_STATE %
%   N9:122  GETTER_PURIFYING %
%   I:5.2  GET_PH_GAS_TC  "TC-3" %
%   N18:15  GETTER_SS_BEGIN_TEMP %
%   N9:121  GETTER_SOFTSTART %
% Rung: 13 %
% TITLE: SOFTSTART LOGIC %
SOR EQU N23:0 N9:121 ONS B29:0/5 MOV 25 N23:14 EOR
%   N23:0  GET_1_STATE %
%   N9:121  GETTER_SOFTSTART %
%   B29:0/5  GET_1_INIT_SOFTSTART %
%   N23:14  GET_1_PH_SS_OUTPUT %

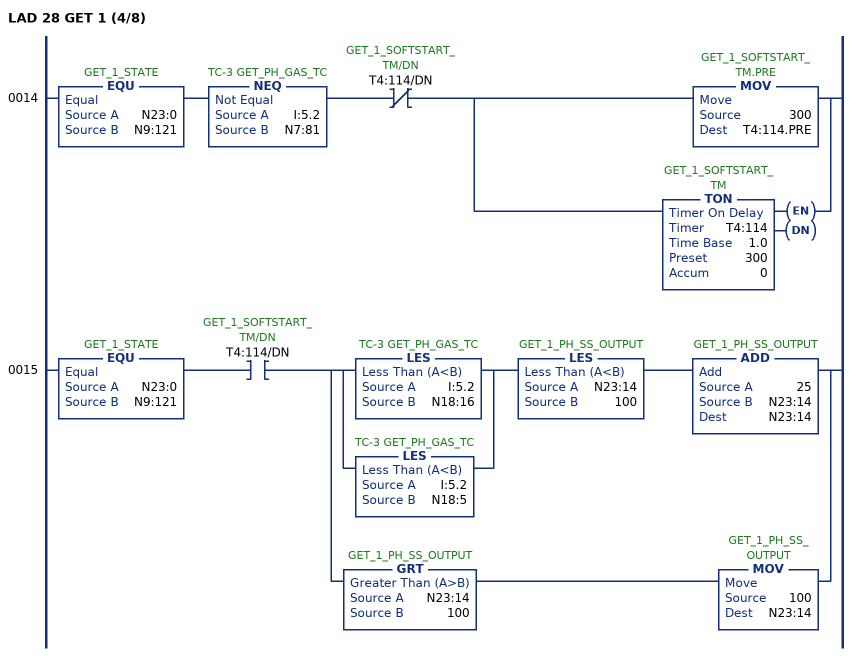
% Rung: 14 %
SOR EQU N23:0 N9:121 NEQ I:5.2 N7:81 XIO T4:114/DN BST MOV 300 T4:114.PRE NXB TON T4:114 1.0 300 0 BND EOR
%   N23:0  GET_1_STATE %
%   N9:121  GETTER_SOFTSTART %
%   I:5.2  GET_PH_GAS_TC  "TC-3" %
%   N7:81  TC_OPEN_SP  "CONFIG The value read by an open TC input" %
%   T4:114  GET_1_SOFTSTART_TM %
% Rung: 15 %
SOR EQU N23:0 N9:121 XIC T4:114/DN BST BST LES I:5.2 N18:16 NXB LES I:5.2 N18:5 BND LES N23:14 100 ADD 25 N23:14 N23:14 NXB GRT N23:14 100 MOV 100 N23:14 BND EOR
%   N23:0  GET_1_STATE %
%   N9:121  GETTER_SOFTSTART %
%   T4:114  GET_1_SOFTSTART_TM %
%   I:5.2  GET_PH_GAS_TC  "TC-3" %
%   N18:16  GETTER_SS_END_TEMP %
%   N18:5  GETTER_PH_SP %
%   N23:14  GET_1_PH_SS_OUTPUT %

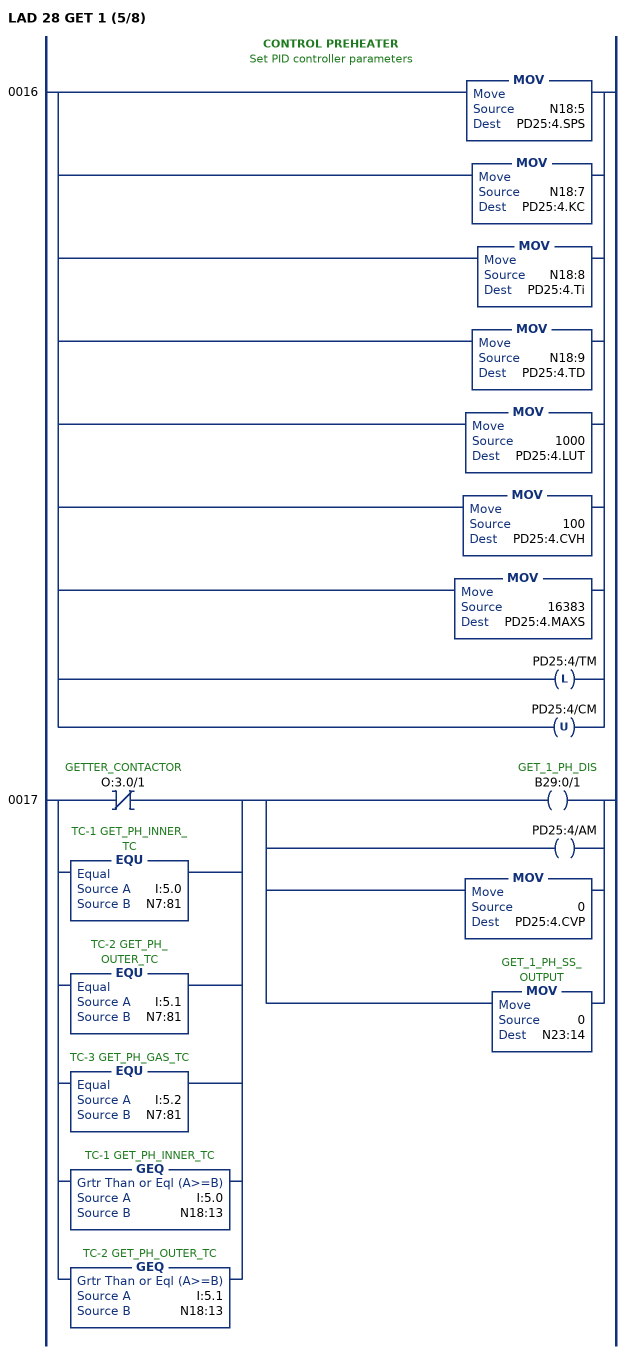
% Rung: 16 %
% TITLE: CONTROL PREHEATER %
% Set PID controller parameters %
SOR BST MOV N18:5 PD25:4.SPS NXB MOV N18:7 PD25:4.KC NXB MOV N18:8 PD25:4.Ti NXB MOV N18:9 PD25:4.TD NXB MOV 1000 PD25:4.LUT NXB MOV 100 PD25:4.CVH NXB MOV 16383 PD25:4.MAXS NXB OTL PD25:4/TM NXB OTU PD25:4/CM BND EOR
%   N18:5  GETTER_PH_SP %
%   N18:7  GET_PH_PID_GAIN %
%   N18:8  GET_PH_PID_INTEG %
%   N18:9  GET_PH_PID_DERIV %
% Rung: 17 %
SOR BST XIO O:3.0/1 NXB EQU I:5.0 N7:81 NXB EQU I:5.1 N7:81 NXB EQU I:5.2 N7:81 NXB GEQ I:5.0 N18:13 NXB GEQ I:5.1 N18:13 BND BST OTE B29:0/1 NXB OTE PD25:4/AM NXB MOV 0 PD25:4.CVP NXB MOV 0 N23:14 BND EOR
%   O:3.0/1  GETTER_CONTACTOR %
%   I:5.0  GET_PH_INNER_TC  "TC-1" %
%   N7:81  TC_OPEN_SP  "CONFIG The value read by an open TC input" %
%   I:5.1  GET_PH_OUTER_TC  "TC-2" %
%   I:5.2  GET_PH_GAS_TC  "TC-3" %
%   N18:13  GET_PH_ROD_LIMIT %
%   B29:0/1  GET_1_PH_DIS %
%   N23:14  GET_1_PH_SS_OUTPUT %

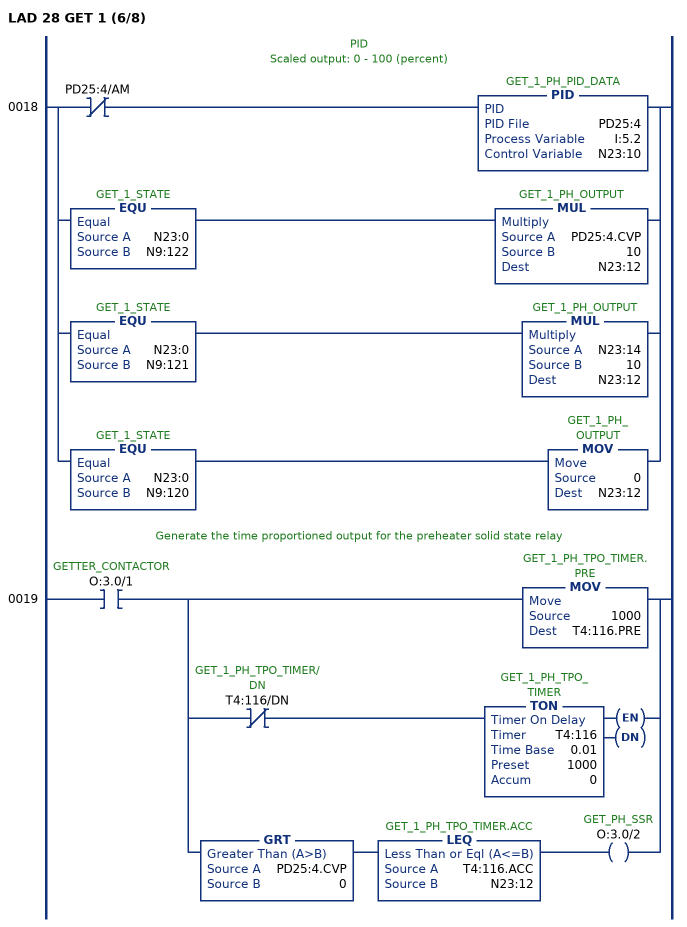
% Rung: 18 %
% PID
% Scaled output: 0 - 100 (percent) %
SOR BST XIO PD25:4/AM PID PD25:4 I:5.2 N23:10 NXB EQU N23:0 N9:122 MUL PD25:4.CVP 10 N23:12 NXB EQU N23:0 N9:121 MUL N23:14 10 N23:12 NXB EQU N23:0 N9:120 MOV 0 N23:12 BND EOR
%   PD25:4  GET_1_PH_PID_DATA %
%   I:5.2  GET_PH_GAS_TC  "TC-3" %
%   N23:10  GET_1_PH_OUT_RAW %
%   N23:0  GET_1_STATE %
%   N9:122  GETTER_PURIFYING %
%   N23:12  GET_1_PH_OUTPUT %
%   N9:121  GETTER_SOFTSTART %
%   N23:14  GET_1_PH_SS_OUTPUT %
%   N9:120  GETTER_STANDBY %
% Rung: 19 %
% Generate the time proportioned output for the preheater solid state relay %
SOR XIC O:3.0/1 BST MOV 1000 T4:116.PRE NXB XIO T4:116/DN TON T4:116 0.01 1000 0 NXB GRT PD25:4.CVP 0 LEQ T4:116.ACC N23:12 OTE O:3.0/2 BND EOR
%   O:3.0/1  GETTER_CONTACTOR %
%   T4:116  GET_1_PH_TPO_TIMER %
%   N23:12  GET_1_PH_OUTPUT %
%   O:3.0/2  GET_PH_SSR %

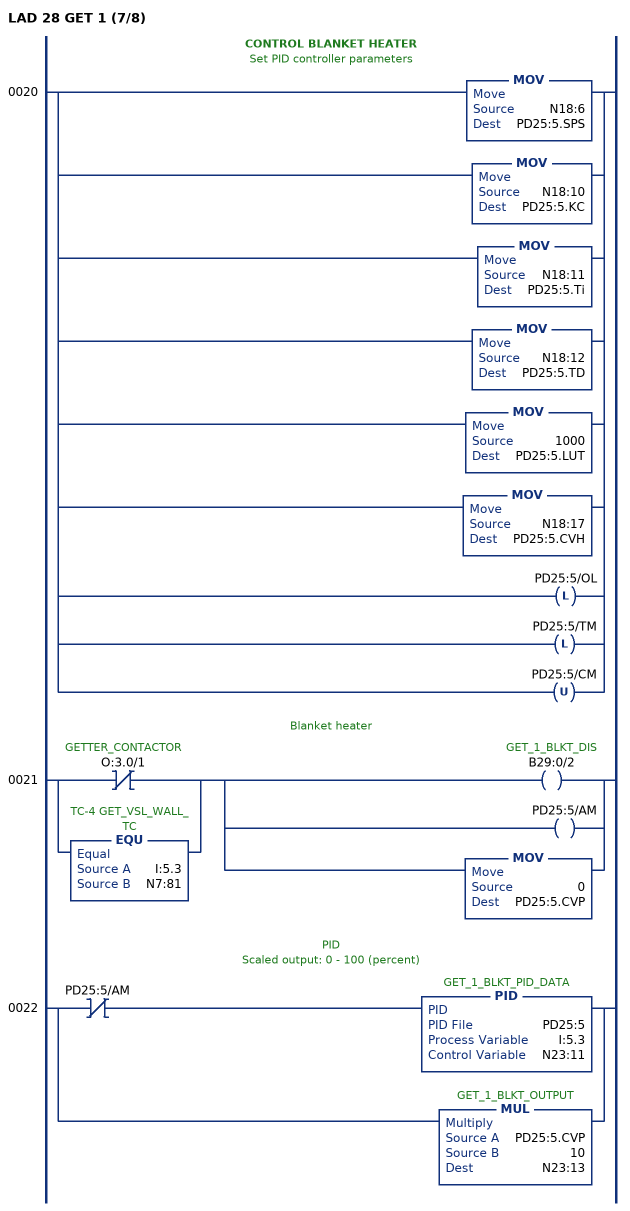
% Rung: 20 %
% TITLE: CONTROL BLANKET HEATER %
% Set PID controller parameters %
SOR BST MOV N18:6 PD25:5.SPS NXB MOV N18:10 PD25:5.KC NXB MOV N18:11 PD25:5.Ti NXB MOV N18:12 PD25:5.TD NXB MOV 1000 PD25:5.LUT NXB MOV N18:17 PD25:5.CVH NXB OTL PD25:5/OL NXB OTL PD25:5/TM NXB OTU PD25:5/CM BND EOR
%   N18:6  GETTER_BLKT_SP %
%   N18:10  GET_BLKT_PID_GAIN %
%   N18:11  GET_BLKT_PID_INTEG %
%   N18:12  GET_BLKT_PID_DERIV %
%   N18:17  GET_BLKT_PID_HI_LIM %
% Rung: 21 %
% Blanket heater %
SOR BST XIO O:3.0/1 NXB EQU I:5.3 N7:81 BND BST OTE B29:0/2 NXB OTE PD25:5/AM NXB MOV 0 PD25:5.CVP BND EOR
%   O:3.0/1  GETTER_CONTACTOR %
%   I:5.3  GET_VSL_WALL_TC  "TC-4" %
%   N7:81  TC_OPEN_SP  "CONFIG The value read by an open TC input" %
%   B29:0/2  GET_1_BLKT_DIS %
% Rung: 22 %
% PID
% Scaled output: 0 - 100 (percent) %
SOR BST XIO PD25:5/AM PID PD25:5 I:5.3 N23:11 NXB MUL PD25:5.CVP 10 N23:13 BND EOR
%   PD25:5  GET_1_BLKT_PID_DATA %
%   I:5.3  GET_VSL_WALL_TC  "TC-4" %
%   N23:11  GET_1_BLKT_OUT_RAW %
%   N23:13  GET_1_BLKT_OUTPUT %

